Fanuc TP program (LS listing): T1_DET_LOST.LS

/PROG  T1_DET_LOST
/ATTR
OWNER		= MNEDITOR;
COMMENT		= "";
PROG_SIZE	= 144;
CREATE		= DATE 25-05-27  TIME 12:39:56;
MODIFIED	= DATE 25-07-16  TIME 19:07:38;
FILE_NAME	= ;
VERSION		= 0;
LINE_COUNT	= 1;
MEMORY_SIZE	= 512;
PROTECT		= READ_WRITE;
TCD:  STACK_SIZE	= 0,
      TASK_PRIORITY	= 50,
      TIME_SLICE	= 0,
      BUSY_LAMP_OFF	= 0,
      ABORT_REQUEST	= 0,
      PAUSE_REQUEST	= 0;
DEFAULT_GROUP	= *,*,*,*,*;
CONTROL_CODE	= 00000000 00000000;
/MN
   1:  UALM[3] ;
/POS
/END
